{attribute 'qualified_only'}
{attribute 'strict'}
{attribute 'to_string'}
TYPE OperationMode :
(
	Manual := 0,
	Recipe := 1,
	Priority := 2
);
END_TYPE

(* stored: Version 1.1.0.1, ProductVersion 3.1.4026.11
   DUT OperationMode: Id {c75456ad-80d1-4040-acf7-93eb29e90b92} *)
